# B&R Automation Studio project AS-lab-1
Automation Studio 

## Logical view

### Library Logical/Libraries/MotorCtrl

#### MotorCtrl.fun
```iecst
FUNCTION_BLOCK FB_Regulator
	VAR_INPUT
		e : REAL;
		e_prev : REAL;
	END_VAR
	VAR_OUTPUT
		u : REAL;
	END_VAR
	VAR
		u_raw : REAL;
		k_p : REAL;
		k_i : REAL;
		integrator : FB_Integrator;
		iyOld : REAL;
		max_abs_value : REAL;
	END_VAR
END_FUNCTION_BLOCK

FUNCTION_BLOCK FB_Motor
	VAR_INPUT
		u : REAL;
	END_VAR
	VAR_OUTPUT
		w : REAL;
		phi : REAL;
	END_VAR
	VAR
		integrator : FB_Integrator;
		integrator_phi : FB_Integrator;
		Tm : REAL;
		ke : REAL;
		enable_reg : BOOL;
	END_VAR
END_FUNCTION_BLOCK

FUNCTION_BLOCK FB_Integrator
	VAR_INPUT
		in : REAL;
	END_VAR
	VAR_OUTPUT
		out : REAL;
	END_VAR
	VAR
		dt : REAL;
		direct : BOOL;
	END_VAR
END_FUNCTION_BLOCK
```

#### FB_Integrator.c
```c
#include <bur/plctypes.h>
#ifdef __cplusplus
	extern "C"
	{
#endif
#include "MotorCtrl.h"
#ifdef __cplusplus
	};
#endif
/* TODO: Add your comment here */
void FB_Integrator(struct FB_Integrator* inst)
{
	inst->out += inst->in * inst->dt;
}
```

#### FB_Motor.c
```c
#include <bur/plctypes.h>
#ifdef __cplusplus
	extern "C"
	{
#endif
#include "MotorCtrl.h"
#ifdef __cplusplus
	};
#endif
/* TODO: Add your comment here */
void FB_Motor(struct FB_Motor* inst)
{
	inst->w = inst->w * inst->Tm / (inst->Tm + inst->dt) +
		inst->u * inst->dt / (inst->ke * (inst->Tm + inst->dt));

	inst->integrator.in = inst->w;
	FB_Integrator(&inst->integrator);
	inst->phi = inst->integrator.out;
}
```

#### FB_Regulator.c
```c
#include <bur/plctypes.h>
#ifdef __cplusplus
	extern "C"
	{
#endif
#include "MotorCtrl.h"
#ifdef __cplusplus
	};
#endif
/* TODO: Add your comment here */
void FB_Regulator(struct FB_Regulator* inst)
{
	/*if (inst->direct)  //direct circuit
	{
		inst->u += (inst->k_p * inst->e <= inst->max_abs_value ? inst->k_p * inst->e : inst->max_abs_value) +
			inst->k_i * inst->dt * inst->e_prev -
			(inst->k_p * inst->e_prev <= inst->max_abs_value ? inst->k_p * inst->e_prev : inst->max_abs_value);

		//truncating output in case it exceeds max. voltage
		if (inst->u > inst->max_abs_value)
			inst->u = inst->max_abs_value;
	}
	else  //feedback circuit
	{
		inst->u_raw = (inst->k_p * inst->e <= inst->max_abs_value ? inst->k_p * inst->e : inst->max_abs_value) -
			(inst->k_p * inst->e_prev <= inst->max_abs_value ? inst->k_p * inst->e_prev : inst->max_abs_value) +
			inst->k_i * inst->dt * inst->e + (inst->u - inst->iyOld);  //right part of the equation

		if (inst->u_raw <= inst->max_abs_value)
			inst->u = inst->u_raw;
		else
		{
			inst->u_raw = (inst->u_raw + inst->max_abs_value) / 2;  //truncating-scheme input
			inst->u = inst->max_abs_value;
		}
		inst->iyOld = inst->u - inst->u_raw;  //updating old truncating-scheme output
	}*/

	if (inst->integrator.direct)
		inst->integrator.in = inst->k_i * inst->e_prev + inst->iyOld / inst->dt;
	else
		inst->integrator.in = inst->k_i * inst->e + inst->iyOld / inst->dt;
	FB_Integrator(&inst->integrator);
	inst->u_raw = (inst->k_p * inst->e <= inst->max_abs_value ? inst->k_p * inst->e : inst->max_abs_value) +
		inst->integrator.out;
	inst->u = inst->u_raw < inst->max_abs_value ? inst->u_raw : inst->max_abs_value;
	inst->iyOld = inst->u - inst->u_raw;
}
```

### Program Logical/Prog1

#### Variables.var
```iecst
VAR
	speed : REAL;
	enable : BOOL;
	motors : ARRAY[0..1] OF FB_Motor;
	regulators : ARRAY[0..1] OF FB_Regulator;
	reg_prevs : ARRAY[0..1] OF REAL;
	mot_prevs : ARRAY[0..1] OF REAL;
END_VAR
```

#### Main.c
```c
#include <bur/plctypes.h>

#ifdef _DEFAULT_INCLUDES
	#include <AsDefault.h>
#endif

void _INIT ProgramInit(void)
{
	//state variables
	enable = count = 0;

	//setting
	speed = 60;

	//regulator
	regulators[0].integrator.dt = 0.002;
	regulators[0].k_p = 0.0064;
	regulators[0].k_i = 0.16;
	regulators[0].max_abs_value = 24;

	//1st motor
	motors[0].integrator.dt = motors[0].integrator_phi.dt = regulators[0].integrator.dt;
	motors[0].Tm = regulators[0].k_p / regulators[0].k_i;
	motors[0].ke = 3 * motors[0].integrator.dt * regulators[0].k_i;
	motors[0].enable_reg = 1;

	//2nd motor
	motors[1].integrator.dt = motors[1].integrator_phi.dt = motors[0].integrator.dt;
	motors[1].Tm = motors[0].Tm;
	motors[1].ke = motors[0].ke;
	motors[1].enable_reg = 0;

	//integrators' structure
	motors[0].integrator.direct = motors[0].integrator_phi.direct = regulators[0].integrator.direct =
		motors[1].integrator.direct = motors[1].integrator_phi.direct = 1;
}

void _CYCLIC ProgramCyclic(void)
{
	//switching system state
	if (count % 100 == 0)
		enable = !enable;

	//switching input
	if (enable)
		speed = 60;
	else
		speed = 0;

	//updating system states
	int i;
	for (i = 0; i < 2; i++)
	{
		if (motors[i].enable_reg)
		{
			//motor with regulator
			regulators[i].e = speed - motors[i].w;
			regulators[i].e_prev = reg_prevs[i];
			FB_Regulator(&regulators[i]);
			motors[i].u = motors[i].integrator.direct ? mot_prevs[i] : regulators[i].u;
			FB_Motor(&motors[i]);

			reg_prevs[i] = regulators[i].e;  //updating previous inputs
			mot_prevs[i] = regulators[i].u;
		}
		else
		{
			//motor without regulator
			motors[i].u = motors[i].integrator.direct ? mot_prevs[i] : speed * motors[i].ke;
			FB_Motor(&motors[i]);

			mot_prevs[i] = speed * motors[i].ke;  //updating previous inputs
		}
	}

	//updating state
	count++;
}

void _EXIT ProgramExit(void)
{

}
```
